{attribute addProperty BoxType "ELX9560-0000-0016"}
{attribute addProperty Id "Power_OKAT %I*BOOL81"}
{attribute addProperty CRC "843727106"}
{attribute addProperty SizeInBites "8"}
{attribute addProperty SizeInBytes "1"}
TYPE Status_Uin_324A4102 :
STRUCT
	{attribute addProperty Name "Power_OK"}
	Power_OK AT %I* : BOOL;
END_STRUCT
END_TYPE

(* stored: Version 1.2.0.0, ProductVersion 3.1.4024.9
   DUT Status_Uin_324A4102: Id {3418e287-c540-4e75-a5f8-0d2a6b4e6aa9} *)
